# B&R Automation Studio project Axis-motion-software-with-endstops
Automation Studio 

## Logical view

### Global.var
```iecst
VAR
	gAxis_X : ACP10AXIS_typ := (0);
	gAxis_X_HW : SdcHwCfg_typ := (0);
	gAxis_X_DrvIf : SdcDrvIf16_typ := (0);
	gAxis_X_DiDoIf : SdcDiDoIf_typ := (0);
	gAxis_X_EncIf : SdcEncIf16_typ := (0);
END_VAR
```
